Yaskawa INFORM job: AAA.JBI

/JOB
//NAME AAA
//POS
///NPOS 102,0,0,0,0,0
///TOOL 11
///POSTYPE PULSE
///PULSE
C00000=-68364,-18948,-30230,-8412,-64593,77319
C00001=-68364,-18948,-30230,-8412,-64593,77319
C00002=-69647,-31187,-44277,-20288,-69402,74286
C00003=-69450,-32025,-45343,-20971,-69925,73655
C00004=-69102,-32717,-46209,-21430,-70532,72890
C00005=-68697,-33336,-46983,-21868,-71169,72094
C00006=-68295,-33928,-47729,-22351,-71811,71308
C00007=-67895,-34507,-48456,-22885,-72449,70538
C00008=-67493,-35080,-49167,-23462,-73081,69784
C00009=-67082,-35642,-49854,-24061,-73707,69040
C00010=-66647,-36180,-50509,-24674,-74322,68302
C00011=-66188,-36704,-51133,-25290,-74928,67571
C00012=-65704,-37217,-51730,-25911,-75522,66847
C00013=-65197,-37724,-52305,-26533,-76098,66135
C00014=-64663,-38231,-52862,-27161,-76651,65437
C00015=-64109,-38751,-53407,-27795,-77179,64756
C00016=-63536,-39287,-53944,-28430,-77681,64092
C00017=-62936,-39841,-54473,-29068,-78149,63446
C00018=-62308,-40407,-54989,-29699,-78588,62814
C00019=-61652,-40985,-55487,-30321,-78998,62197
C00020=-60960,-41567,-55961,-30929,-79380,61590
C00021=-60233,-42148,-56410,-31512,-79742,60992
C00022=-59467,-42711,-56818,-32075,-80077,60402
C00023=-58661,-43256,-57185,-32608,-80396,59817
C00024=-57815,-43767,-57504,-33108,-80699,59237
C00025=-56929,-44245,-57773,-33585,-80981,58663
C00026=-56004,-44691,-57993,-34026,-81256,58093
C00027=-55042,-45096,-58164,-34439,-81514,57528
C00028=-54041,-45462,-58282,-34825,-81757,56968
C00029=-53009,-45783,-58352,-35183,-81986,56416
C00030=-51941,-46064,-58372,-35510,-82208,55867
C00031=-50837,-46287,-58316,-35814,-82415,55324
C00032=-49706,-46480,-58249,-36089,-82606,54790
C00033=-48543,-46623,-58125,-36336,-82793,54261
C00034=-47352,-46712,-57942,-36561,-82962,53740
C00035=-46132,-46761,-57717,-36756,-83128,53224
C00036=-44885,-46753,-57442,-36926,-83284,52716
C00037=-43609,-46702,-57126,-37071,-83426,52215
C00038=-42313,-46606,-56756,-37190,-83564,51721
C00039=-40992,-46469,-56353,-37283,-83694,51235
C00040=-39642,-46286,-55906,-37348,-83815,50755
C00041=-38274,-46058,-55417,-37389,-83923,50285
C00042=-36881,-45778,-54880,-37402,-84030,49822
C00043=-35461,-45466,-54313,-37380,-84133,49363
C00044=-34021,-45089,-53690,-37333,-84227,48915
C00045=-32556,-44667,-53026,-37253,-84327,48471
C00046=-31068,-44186,-52314,-37137,-84427,48034
C00047=-29549,-43643,-51551,-36985,-84532,47600
C00048=-28006,-43036,-50736,-36795,-84642,47172
C00049=-26438,-42365,-49870,-36567,-84764,46750
C00050=-24843,-41624,-48950,-36298,-84894,46332
C00051=-23218,-40828,-47982,-35987,-85044,45916
C00052=-21567,-39963,-46963,-35636,-85195,45508
C00053=-19890,-39047,-45902,-35241,-85362,45104
C00054=-18183,-38071,-44792,-34801,-85546,44705
C00055=-16444,-37041,-43641,-34314,-85739,44311
C00056=-14675,-35962,-42450,-33780,-85942,43922
C00057=-12875,-34828,-41218,-33194,-86164,43538
C00058=-11039,-33639,-39945,-32556,-86404,43158
C00059=-9168,-32399,-38636,-31863,-86666,42781
C00060=-7260,-31087,-37277,-31115,-86948,42407
C00061=-5317,-29712,-35879,-30310,-87260,42037
C00062=-3335,-28272,-34442,-29448,-87602,41669
C00063=-1314,-26758,-32963,-28529,-87978,41302
C00064=740,-25180,-31454,-27554,-88397,40937
C00065=2830,-23535,-29912,-26525,-88845,40575
C00066=4955,-21815,-28343,-25442,-89330,40215
C00067=7110,-20037,-26756,-24311,-89858,39857
C00068=9296,-18201,-25165,-23135,-90424,39499
C00069=11500,-16314,-23574,-21922,-91025,39147
C00070=13724,-14357,-21976,-20674,-91664,38795
C00071=15960,-12340,-20385,-19402,-92347,38444
C00072=18201,-10264,-18809,-18114,-93070,38094
C00073=20439,-8128,-17251,-16820,-93839,37744
C00074=22660,-5921,-15710,-15533,-94646,37394
C00075=24861,-3660,-14198,-14261,-95504,37041
C00076=27031,-1318,-12703,-13017,-96403,36684
C00077=29160,1095,-11231,-11811,-97349,36323
C00078=31238,3581,-9790,-10658,-98341,35956
C00079=33256,6152,-8360,-9564,-99378,35582
C00080=35212,8796,-6953,-8541,-100468,35196
C00081=37090,11539,-5562,-7600,-101601,34798
C00082=38890,14357,-4182,-6748,-102784,34386
C00083=40606,17247,-2830,-5987,-103989,33962
C00084=42234,20176,-1515,-5328,-105226,33522
C00085=43779,23147,-231,-4766,-106475,33067
C00086=45236,26126,1005,-4303,-107723,32599
C00087=46613,29101,2179,-3939,-108966,32116
C00088=47910,32075,3307,-3674,-110201,31618
C00089=49120,35066,4387,-3510,-111426,31104
C00090=50253,38065,5432,-3448,-112654,30569
C00091=51303,41052,6424,-3500,-113871,30014
C00092=52280,44039,7368,-3653,-115079,29436
C00093=53181,46996,8251,-3901,-116245,28843
C00094=54021,49888,9056,-4252,-117382,28229
C00095=54794,52744,9798,-4694,-118477,27598
C00096=55513,55553,10477,-5230,-119542,26946
C00097=56178,58291,11079,-5846,-120549,26281
C00098=56813,60861,11556,-6511,-121443,25623
C00099=57429,63293,11953,-7215,-122251,24970
C00100=57972,65908,12380,-8063,-123164,24251
C00101=62816,85729,13832,-16988,-127514,18274
//INST
///DATE 2023/06/21 17:13
///ATTR SC,RW
///GROUP1 RB1
NOP
MOVJ C00000 VJ=5.0
TIMER T=1.00
MOVJ C00001 VJ=1.0
TIMER T=0.10
MOVL C00002 V=300.0
MOVL C00003 V=300.0
MOVL C00004 V=300.0
MOVL C00005 V=300.0
MOVL C00006 V=300.0
MOVL C00007 V=300.0
MOVL C00008 V=300.0
MOVL C00009 V=300.0
MOVL C00010 V=300.0
MOVL C00011 V=300.0
MOVL C00012 V=300.0
MOVL C00013 V=300.0
MOVL C00014 V=300.0
MOVL C00015 V=300.0
MOVL C00016 V=300.0
MOVL C00017 V=300.0
MOVL C00018 V=300.0
MOVL C00019 V=300.0
MOVL C00020 V=300.0
MOVL C00021 V=300.0
MOVL C00022 V=300.0
MOVL C00023 V=300.0
MOVL C00024 V=300.0
MOVL C00025 V=300.0
MOVL C00026 V=300.0
MOVL C00027 V=300.0
MOVL C00028 V=300.0
MOVL C00029 V=300.0
MOVL C00030 V=300.0
MOVL C00031 V=300.0
MOVL C00032 V=300.0
MOVL C00033 V=300.0
MOVL C00034 V=300.0
MOVL C00035 V=300.0
MOVL C00036 V=300.0
MOVL C00037 V=300.0
MOVL C00038 V=300.0
MOVL C00039 V=300.0
MOVL C00040 V=300.0
MOVL C00041 V=300.0
MOVL C00042 V=300.0
MOVL C00043 V=300.0
MOVL C00044 V=300.0
MOVL C00045 V=300.0
MOVL C00046 V=300.0
MOVL C00047 V=300.0
MOVL C00048 V=300.0
MOVL C00049 V=300.0
MOVL C00050 V=300.0
MOVL C00051 V=300.0
MOVL C00052 V=300.0
MOVL C00053 V=300.0
MOVL C00054 V=300.0
MOVL C00055 V=300.0
MOVL C00056 V=300.0
MOVL C00057 V=300.0
MOVL C00058 V=300.0
MOVL C00059 V=300.0
MOVL C00060 V=300.0
MOVL C00061 V=300.0
MOVL C00062 V=300.0
MOVL C00063 V=300.0
MOVL C00064 V=300.0
MOVL C00065 V=300.0
MOVL C00066 V=300.0
MOVL C00067 V=300.0
MOVL C00068 V=300.0
MOVL C00069 V=300.0
MOVL C00070 V=300.0
MOVL C00071 V=300.0
MOVL C00072 V=300.0
MOVL C00073 V=300.0
MOVL C00074 V=300.0
MOVL C00075 V=300.0
MOVL C00076 V=300.0
MOVL C00077 V=300.0
MOVL C00078 V=300.0
MOVL C00079 V=300.0
MOVL C00080 V=300.0
MOVL C00081 V=300.0
MOVL C00082 V=300.0
MOVL C00083 V=300.0
MOVL C00084 V=300.0
MOVL C00085 V=300.0
MOVL C00086 V=300.0
MOVL C00087 V=300.0
MOVL C00088 V=300.0
MOVL C00089 V=300.0
MOVL C00090 V=300.0
MOVL C00091 V=300.0
MOVL C00092 V=300.0
MOVL C00093 V=300.0
MOVL C00094 V=300.0
MOVL C00095 V=300.0
MOVL C00096 V=300.0
MOVL C00097 V=300.0
MOVL C00098 V=300.0
MOVL C00099 V=300.0
MOVL C00100 V=300.0
MOVL C00101 V=300.0
END
